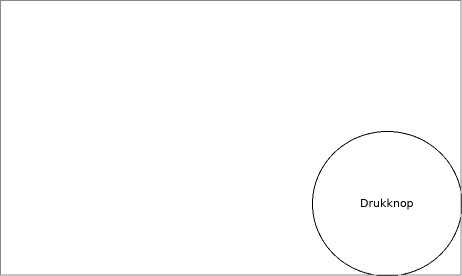
VISUALIZATION Visualization_GetMinimumClicker  // 462x276
    Ellipse (312,131 150x145), "Drukknop"
        tap prg_GetMinimum.bDrukknop
END_VISUALIZATION

(* stored: Version 1.1.0.1, ProductVersion 3.1.4024.15
   Visu Visualization_GetMinimumClicker: Id {4a722c4c-3378-46a8-b901-0257e0fa2c4c} *)
